PROGRAM commit1
VAR
END_VAR

END_PROGRAM

(* stored: Version 1.1.0.1, ProductVersion 3.1.4024.12
   POU commit1: Id {b514ab45-b3b1-4c4e-b7a4-8ac05743b23d}, SpecialFunc None *)
